// TIA Portal V20 export
DATA_BLOCK "OtherSafetyInterface"   // DB211
// stored: MemoryReserve 100
   VAR
      OtherDoor1 : "LER_typefDoorInterface";   // BA010 Other Door
      OtherDoor2 : "LER_typefDoorInterface";   // BA015 Other Door
      OtherDoor3 : "LER_typefDoorInterface";   // BA030 Other Door
      OtherDoor4 : "LER_typefDoorInterface";   // BA060 Other Door
      InspectionExternalDoor { S7_SetPoint := 'True'} : "LER_typefDoorInterface";   // Inspection External Door
      Inspection30MaintDoor { S7_SetPoint := 'True'} : "LER_typefDoorInterface";   // Inspection BA030 Main Door
      Inspection40MaintDoor { S7_SetPoint := 'True'} : "LER_typefDoorInterface";   // Inspection BA040 Main Door
      OtherEMO1 { S7_SetPoint := 'True'} : Bool;   // BA010 EMO
      OtherEMO2 { S7_SetPoint := 'True'} : Bool;   // BA015 EMO
      OtherEMO3 { S7_SetPoint := 'True'} : Bool;   // BA030 EMO
      OtherEMO4 { S7_SetPoint := 'True'} : Bool;   // BA060 EMO
      Inspection30LightCurtain { S7_SetPoint := 'True'} : "LER_typeLightCurtainInterface";   // BA060 Stack #1 Light Curatain
      Inspection40LightCurtain { S7_SetPoint := 'True'} : "LER_typeLightCurtainInterface";   // BA060 Stack #2 Light Curatain
      "30CathodeConveyorCover" { S7_SetPoint := 'True'} : "LER_typeConveyorCoverInterface";   // BA030 Cathode Conveyor Cover
      "30AnodeConveyorCover" { S7_SetPoint := 'True'} : "LER_typeConveyorCoverInterface";   // BA030 Cathode Anode Cover
      "40CathodeConveyorCover" { S7_SetPoint := 'True'} : "LER_typeConveyorCoverInterface";   // BA040 Cathode Conveyor Cover
      "40AnodeConveyorCover" { S7_SetPoint := 'True'} : "LER_typeConveyorCoverInterface";   // BA040 Cathode Anode Cover
   END_VAR
BEGIN
   OtherDoor1.configuration.referenceDesignator := WSTRING#'10';
   OtherDoor2.configuration.referenceDesignator := WSTRING#'15';
   OtherDoor3.configuration.referenceDesignator := WSTRING#'30';
   OtherDoor4.configuration.referenceDesignator := WSTRING#'60';
   InspectionExternalDoor.configuration.referenceDesignator := WSTRING#'60';
   Inspection30MaintDoor.configuration.referenceDesignator := WSTRING#'30';
   Inspection40MaintDoor.configuration.referenceDesignator := WSTRING#'40';
   Inspection30LightCurtain.configuration.referenceDesignator := WSTRING#'30';
   Inspection40LightCurtain.configuration.referenceDesignator := WSTRING#'40';
   "30CathodeConveyorCover".configuration.referenceDesignator := WSTRING#'30-CA';
   "30AnodeConveyorCover".configuration.referenceDesignator := WSTRING#'30-AN';
   "40CathodeConveyorCover".configuration.referenceDesignator := WSTRING#'40-CA';
   "40AnodeConveyorCover".configuration.referenceDesignator := WSTRING#'40-AN';
END_DATA_BLOCK
